PROGRAM PRG_1
VAR
	sLog : STRING;
END_VAR

sLog := 'Hi, there!';

END_PROGRAM

(* stored: Version 1.1.0.1, ProductVersion 3.1.4024.16
   POU PRG_1: Id {6c9bef0d-f3e5-45c1-b5f7-36d7b9cf93d7}, SpecialFunc None *)
